(* IEC 61131-3 sources: Structured-Text/Source Code/Utility/FLASHER, 2 files *)

(* ---- FLASHER.ST ---- *)
//Generates an On/Off pattern when the input is on.

RSA(SET := IN, RESET1 := TON_2.Q);
TON_1(IN := RSA.Q1, PT := PT_ON);
TON_2(IN := TON_1.Q, PT := PT_OFF);

//Set Output.
IF IN AND NOT TON_1.Q THEN
	OUT := TRUE;
ELSE
	OUT := FALSE;
END_IF;

(* ---- Local Variables.ST ---- *)
VAR_INPUT
	IN:		BOOL;
	PT_ON:	TIME;
	PT_OFF:	TIME;
END_VAR

VAR_OUTPUT
	OUT:	BOOL;
END_VAR

VAR
	TON_1:	TON;
	TON_2:	TON;
	RSA:	RS;
END_VAR
